(* IEC 61131-3 sources: com.logicals.lc3.webinar/usRTS_RPMControl_iSOC/src_FB_LIB_SAFE/Counter/DINT, 3 files *)

(* ---- wCTD_DINT.iecst ---- *)
NAMESPACE logicals.web.standard
NAMESPACE counter

/*
 * Function block wrapper for IEC 61131-3 CTD_DINT<br>
 * CD = decrement on positive edge on CD (BOOL)<br>
 * LD = flag for reset (CV:=PV) (BOOL)<br>
 * PV = initial value for counting (DINT)<br>
 * Q  = flag showing whether 0 is reached or not (BOOL)<br>
 * CV = current value of counter (DINT)<br>
 */
FUNCTION_BLOCK wCTD_DINT
	{ CV { index := 2 }; vNameAlignment:="center"; altName:="CTD_DINT"; bgColor:="LightPink"; width:=120; }
	VAR_INPUT
		CD : BOOL /* R_EDGE */;
		LD : BOOL;
		PV : DINT;
	END_VAR
	VAR_OUTPUT
		Q  : BOOL;
		CV : DINT;
	END_VAR
	VAR
		CTD_DINT : CTD_DINT;
	END_VAR

	CTD_DINT(CD:=CD, LD:=LD, PV:=PV, Q=>Q, CV=>CV, ENO=>ENO);
END_FUNCTION_BLOCK

END_NAMESPACE
END_NAMESPACE

(* ---- wCTU_DINT.iecst ---- *)
NAMESPACE logicals.web.standard
NAMESPACE counter

/*
 * Function block wrapper for IEC 61131-3 CTU_DINT<br>
 * CU = increment on positive edge on CU (BOOL)<br>
 * R  = flag for reset (BOOL)<br>
 * PV = upper limit of counter (DINT)<br>
 * Q  = flag showing whether upper limit is reached or not (BOOL)<br>
 * CV = current value of counter (DINT)<br>
 */
FUNCTION_BLOCK wCTU_DINT
	{ CV { index := 2 }; vNameAlignment:="center"; altName:="CTU_DINT"; bgColor:="LightPink"; width:=120; }
	VAR_INPUT
		CU : BOOL /* R_EDGE */;
		R  : BOOL;
		PV : DINT;
	END_VAR
	VAR_OUTPUT
		Q  : BOOL;
		CV : DINT;
	END_VAR
	VAR
		M : BOOL;
	END_VAR
	VAR_TEMP
		edgeCU : BOOL;
	END_VAR

	/* Perform Edge Recognition */
	IF CU THEN
		edgeCU := NOT M;
		M := TRUE;
	ELSE
		edgeCU := CU;
		M := FALSE;
	END_IF;

	IF R THEN
		CV := 0;
	ELSE
		IF edgeCU THEN
			IF CV < 16#7FFFFFFF THEN
				CV := CV + 1;
			END_IF;
		END_IF;
	END_IF;
	Q := CV >= PV;
END_FUNCTION_BLOCK

END_NAMESPACE
END_NAMESPACE

(* ---- wCTUD_DINT.iecst ---- *)
NAMESPACE logicals.web.standard
NAMESPACE counter

/*
 * Function block wrapper for IEC 61131-3 CTUD_DINT<br>
 * CU = increment on positive edge on CU (BOOL)<br>
 * CD = decrement on positive edge on CD (BOOL)<br>
 * R  = flag for reset (CV:=0) (BOOL)<br>
 * LD = flag for load (CV:=PV) (BOOL)<br>
 * PV = upper limit of counter (DINT)<br>
 * QU = flag showing whether upper limit is reached or not (BOOL)<br>
 * QD = flag showing whether 0 is reached or not (BOOL)<br>
 * CV = current value of counter (DINT)<br>
 */
FUNCTION_BLOCK wCTUD_DINT
	{ vNameAlignment:="center"; altName:="CTUD_DINT"; bgColor:="LightPink"; width:=120; }
	VAR_INPUT
		CU : BOOL /* R_EDGE */;
		CD : BOOL /* R_EDGE */;
		R  : BOOL;
		LD : BOOL;
		PV : DINT;
	END_VAR
	VAR_OUTPUT
		QU : BOOL;
		QD : BOOL;
		CV : DINT;
	END_VAR
	VAR
		CTUD_DINT : CTUD_DINT;
	END_VAR

	CTUD_DINT(CU:=CU, CD:=CD, R:=R, LD:=LD, PV:=PV, QU=>QU, QD=>QD, CV=>CV, ENO=>ENO);
END_FUNCTION_BLOCK

END_NAMESPACE
END_NAMESPACE
